(* IEC 61131-3 sources: inproshop/test9_exported/2.Main, 6 files *)

(* ---- Main_Clock.st ---- *)
VAR_GLOBAL
	CPU_Clock:Str_Clock;
END_VAR

(* ---- Main_Communication.st ---- *)
VAR_GLOBAL
	From_OPXX AT %IW2000:Str_OP10_TO_OPXX;
	TO_OPXX AT %QW2000:Str_OPXX_TO_OP10;
	To_Slave:Str_ToSlave;

END_VAR

(* ---- Main_IO.st ---- *)
VAR_GLOBAL

	IX7000_0	AT	%IX7000.0:BOOL;
	IX7000_1	AT	%IX7000.1:BOOL;
	IX7000_2	AT	%IX7000.2:BOOL;
	IX7000_3	AT	%IX7000.3:BOOL;
	IX7000_4	AT	%IX7000.4:BOOL;
	IX7000_5	AT	%IX7000.5:BOOL;
	IX7000_6	AT	%IX7000.6:BOOL;
	IX7000_7	AT	%IX7000.7:BOOL;
	IX7001_0_OP07启动按钮HMI1	AT	%IX7001.0:BOOL;
	IX7001_1_OP07停止按钮HMI1	AT	%IX7001.1:BOOL;
	IX7001_2_OP07复位按钮HMI1	AT	%IX7001.2:BOOL;
	IX7001_3_OP07手自动旋钮HMI1	AT	%IX7001.3:BOOL;
	IX7001_4_OP07急停按钮HMI	AT	%IX7001.4:BOOL;
	IX7001_5_OP07启动按钮左	AT	%IX7001.5:BOOL;
	IX7001_6_OP07停止按钮左	AT	%IX7001.6:BOOL;
	IX7001_7_OP07复位按钮左	AT	%IX7001.7:BOOL;
	IX7002_0_OP07手自动旋钮左	AT	%IX7002.0:BOOL;
	IX7002_1_OP07急停按钮左	AT	%IX7002.1:BOOL;
	IX7002_2_OP07启动按钮右	AT	%IX7002.2:BOOL;
	IX7002_3_OP07停止按钮右	AT	%IX7002.3:BOOL;
	IX7002_4_OP07复位按钮右	AT	%IX7002.4:BOOL;
	IX7002_5_OP07手自动旋钮右	AT	%IX7002.5:BOOL;
	IX7002_6_OP07急停按钮右	AT	%IX7002.6:BOOL;
	IX7002_7_OP07安全门1	AT	%IX7002.7:BOOL;
	IX7003_0_OP07安全门2	AT	%IX7003.0:BOOL;
	IX7003_1_OP07安全门3	AT	%IX7003.1:BOOL;
	IX7003_2_OP07安全门4	AT	%IX7003.2:BOOL;
	IX7003_3_OP07安全门5	AT	%IX7003.3:BOOL;
	IX7003_4_OP07安全门6	AT	%IX7003.4:BOOL;
	IX7003_5_OP07安全门7	AT	%IX7003.5:BOOL;
	IX7003_6_OP07安全门8	AT	%IX7003.6:BOOL;
	IX7003_7	AT	%IX7003.7:BOOL;
	IX7004_0	AT	%IX7004.0:BOOL;
	IX7004_1	AT	%IX7004.1:BOOL;
	IX7004_2	AT	%IX7004.2:BOOL;
	IX7004_3	AT	%IX7004.3:BOOL;
	IX7004_4	AT	%IX7004.4:BOOL;
	IX7004_5	AT	%IX7004.5:BOOL;
	IX7004_6	AT	%IX7004.6:BOOL;
	IX7004_7_水冷机故障	AT	%IX7004.7:BOOL;
	IX7005_0_供钉机1_缺钉报警	AT	%IX7005.0:BOOL;
	IX7005_1_供钉机1_供钉完成	AT	%IX7005.1:BOOL;
	IX7005_2_供钉机1_钉入管检测	AT	%IX7005.2:BOOL;
	IX7005_3_供钉机1_钉到位检测	AT	%IX7005.3:BOOL;
	IX7005_4_电批1_结果OK	AT	%IX7005.4:BOOL;
	IX7005_5_电批1_结果NG	AT	%IX7005.5:BOOL;
	IX7005_6_电批1_ERROR	AT	%IX7005.6:BOOL;
	IX7005_7_电批1_预留	AT	%IX7005.7:BOOL;
	IX7006_0_供钉机2_缺钉报警	AT	%IX7006.0:BOOL;
	IX7006_1_供钉机2_供钉完成	AT	%IX7006.1:BOOL;
	IX7006_2_供钉机2_钉入管检测	AT	%IX7006.2:BOOL;
	IX7006_3_供钉机2_钉到位检测	AT	%IX7006.3:BOOL;
	IX7006_4_电批2_结果OK	AT	%IX7006.4:BOOL;
	IX7006_5_电批2_结果NG	AT	%IX7006.5:BOOL;
	IX7006_6_电批2_ERROR	AT	%IX7006.6:BOOL;
	IX7006_7_电批2_预留	AT	%IX7006.7:BOOL;
	IX7007_0_供钉机3_缺钉报警	AT	%IX7007.0:BOOL;
	IX7007_1_供钉机3_供钉完成	AT	%IX7007.1:BOOL;
	IX7007_2_供钉机3_钉入管检测	AT	%IX7007.2:BOOL;
	IX7007_3_供钉机3_钉到位检测	AT	%IX7007.3:BOOL;
	IX7007_4_电批3_结果OK	AT	%IX7007.4:BOOL;
	IX7007_5_电批3_结果NG	AT	%IX7007.5:BOOL;
	IX7007_6_电批3_ERROR	AT	%IX7007.6:BOOL;
	IX7007_7_电批3_预留	AT	%IX7007.7:BOOL;
	IX7008_0_供钉机4_供钉完成	AT	%IX7008.0:BOOL;
	IX7008_1_供钉机4_预留	AT	%IX7008.1:BOOL;
	IX7008_2_供钉机4_预留	AT	%IX7008.2:BOOL;
	IX7008_3_供钉机4_预留	AT	%IX7008.3:BOOL;
	IX7008_4_电批4_结果OK	AT	%IX7008.4:BOOL;
	IX7008_5_电批4_结果NG	AT	%IX7008.5:BOOL;
	IX7008_6_电批4_ERROR	AT	%IX7008.6:BOOL;
	IX7008_7_电批4_预留	AT	%IX7008.7:BOOL;
	IX7009_0	AT	%IX7009.0:BOOL;
	IX7009_1	AT	%IX7009.1:BOOL;
	IX7009_2	AT	%IX7009.2:BOOL;
	IX7009_3	AT	%IX7009.3:BOOL;
	IX7009_4	AT	%IX7009.4:BOOL;
	IX7009_5	AT	%IX7009.5:BOOL;
	IX7009_6	AT	%IX7009.6:BOOL;
	IX7009_7	AT	%IX7009.7:BOOL;
	IX7100_0_启动按钮1	AT	%IX7100.0:BOOL;
	IX7100_1_启动按钮2	AT	%IX7100.1:BOOL;
	IX7100_2_安全光栅	AT	%IX7100.2:BOOL;
	IX7100_3	AT	%IX7100.3:BOOL;
	IX7100_4_上料1侧边定位气缸CY01_伸出	AT	%IX7100.4:BOOL;
	IX7100_5_上料1侧边定位气缸CY01_缩回	AT	%IX7100.5:BOOL;
	IX7100_6_上料避位升降气缸CY02_上升	AT	%IX7100.6:BOOL;
	IX7100_7_上料避位升降气缸CY02_下降	AT	%IX7100.7:BOOL;
	IX7101_0_物料有无检测Sensor1	AT	%IX7101.0:BOOL;
	IX7101_1_物料有无检测Sensor2	AT	%IX7101.1:BOOL;
	IX7101_2	AT	%IX7101.2:BOOL;
	IX7101_3	AT	%IX7101.3:BOOL;
	IX7101_4	AT	%IX7101.4:BOOL;
	IX7101_5	AT	%IX7101.5:BOOL;
	IX7101_6	AT	%IX7101.6:BOOL;
	IX7101_7	AT	%IX7101.7:BOOL;
	IX7102_0_搬运1_1旋转气缸CY03_放料位	AT	%IX7102.0:BOOL;
	IX7102_1_搬运1_1旋转气缸CY03_取料位	AT	%IX7102.1:BOOL;
	IX7102_2_搬运1_1夹爪气缸CY04_夹紧位	AT	%IX7102.2:BOOL;
	IX7102_3_搬运1_1夹爪气缸CY04_打开位	AT	%IX7102.3:BOOL;
	IX7102_4_搬运1_1避让气缸CY05A_伸出位	AT	%IX7102.4:BOOL;
	IX7102_5_搬运1_1避让气缸CY05A_缩回位	AT	%IX7102.5:BOOL;
	IX7102_6_搬运1_1避让气缸CY05B_伸出位	AT	%IX7102.6:BOOL;
	IX7102_7_搬运1_1避让气缸CY05B_缩回位	AT	%IX7102.7:BOOL;
	IX7103_0_搬运1_2旋转气缸CY06_放料位	AT	%IX7103.0:BOOL;
	IX7103_1_搬运1_2旋转气缸CY06_取料位	AT	%IX7103.1:BOOL;
	IX7103_2_搬运1_2夹爪气缸CY07_夹紧位	AT	%IX7103.2:BOOL;
	IX7103_3_搬运1_2夹爪气缸CY07_打开位	AT	%IX7103.3:BOOL;
	IX7103_4_搬运1_2避让气缸CY08_伸出位	AT	%IX7103.4:BOOL;
	IX7103_5_搬运1_2避让气缸CY08_缩回位	AT	%IX7103.5:BOOL;
	IX7103_6	AT	%IX7103.6:BOOL;
	IX7103_7	AT	%IX7103.7:BOOL;
	IX7104_0_搬运2_1旋转气缸CY09_放料位	AT	%IX7104.0:BOOL;
	IX7104_1_搬运2_1旋转气缸CY09_取料位	AT	%IX7104.1:BOOL;
	IX7104_2_搬运2_1夹爪气缸CY10_夹紧位	AT	%IX7104.2:BOOL;
	IX7104_3_搬运2_1夹爪气缸CY10_打开位	AT	%IX7104.3:BOOL;
	IX7104_4_搬运2_1避让气缸CY11_伸出位	AT	%IX7104.4:BOOL;
	IX7104_5_搬运2_1避让气缸CY11_缩回位	AT	%IX7104.5:BOOL;
	IX7104_6	AT	%IX7104.6:BOOL;
	IX7104_7	AT	%IX7104.7:BOOL;
	IX7105_0_搬运2_2旋转气缸CY12_放料位	AT	%IX7105.0:BOOL;
	IX7105_1_搬运2_2旋转气缸CY12_取料位	AT	%IX7105.1:BOOL;
	IX7105_2_搬运2_2夹爪气缸CY13_夹紧位	AT	%IX7105.2:BOOL;
	IX7105_3_搬运2_2夹爪气缸CY13_打开位	AT	%IX7105.3:BOOL;
	IX7105_4_搬运2_2避让气缸CY14_伸出位	AT	%IX7105.4:BOOL;
	IX7105_5_搬运2_2避让气缸CY14_缩回位	AT	%IX7105.5:BOOL;
	IX7105_6	AT	%IX7105.6:BOOL;
	IX7105_7	AT	%IX7105.7:BOOL;
	IX7106_0_平台1避位升降气缸CY15_上升位	AT	%IX7106.0:BOOL;
	IX7106_1_平台1避位升降气缸CY15_下降位	AT	%IX7106.1:BOOL;
	IX7106_2_平台1侧推定位X气缸CY16_缩回位	AT	%IX7106.2:BOOL;
	IX7106_3_平台1侧推定位X气缸CY16_伸出位	AT	%IX7106.3:BOOL;
	IX7106_4_平台1侧推定位Y气缸CY17_伸出位	AT	%IX7106.4:BOOL;
	IX7106_5_平台1侧推定位Y气缸CY17_缩回位	AT	%IX7106.5:BOOL;
	IX7106_6_平台1物料压紧气缸CY18_下降位	AT	%IX7106.6:BOOL;
	IX7106_7_平台1物料压紧气缸CY18_上升位	AT	%IX7106.7:BOOL;
	IX7107_0_平台1物料有无检测Sensor3	AT	%IX7107.0:BOOL;
	IX7107_1_平台2物料有无检测Sensor4	AT	%IX7107.1:BOOL;
	IX7107_2_平台2避位升降气缸CY19_上升位	AT	%IX7107.2:BOOL;
	IX7107_3_平台2避位升降气缸CY19_下降位	AT	%IX7107.3:BOOL;
	IX7107_4_平台2侧推定位Y气缸CY20_伸出位	AT	%IX7107.4:BOOL;
	IX7107_5_平台2侧推定位Y气缸CY20_缩回位	AT	%IX7107.5:BOOL;
	IX7107_6_平台2物料压紧气缸CY21_下降位	AT	%IX7107.6:BOOL;
	IX7107_7_平台2物料压紧气缸CY21_上升位	AT	%IX7107.7:BOOL;
	IX7108_0_平台3避位升降气缸CY22_上升位	AT	%IX7108.0:BOOL;
	IX7108_1_平台3避位升降气缸CY22_下降位	AT	%IX7108.1:BOOL;
	IX7108_2_平台4侧推定位X气缸CY23_缩回位	AT	%IX7108.2:BOOL;
	IX7108_3_平台4侧推定位X气缸CY23_伸出位	AT	%IX7108.3:BOOL;
	IX7108_4_平台3侧推定位Y气缸CY24_伸出位	AT	%IX7108.4:BOOL;
	IX7108_5_平台3侧推定位Y气缸CY24_缩回位	AT	%IX7108.5:BOOL;
	IX7108_6_平台3物料压紧气缸CY25_下降位	AT	%IX7108.6:BOOL;
	IX7108_7_平台3物料压紧气缸CY25_上升位	AT	%IX7108.7:BOOL;
	IX7109_0_平台3物料有无检测Sensor5	AT	%IX7109.0:BOOL;
	IX7109_1_平台4物料有无检测Sensor6	AT	%IX7109.1:BOOL;
	IX7109_2_平台4避位升降气缸CY26_上升位	AT	%IX7109.2:BOOL;
	IX7109_3_平台4避位升降气缸CY26_下降位	AT	%IX7109.3:BOOL;
	IX7109_4_平台4侧推定位Y气缸CY27_缩回位	AT	%IX7109.4:BOOL;
	IX7109_5_平台4侧推定位Y气缸CY27_伸出位	AT	%IX7109.5:BOOL;
	IX7109_6_平台4物料旋转气缸CY28_下料位	AT	%IX7109.6:BOOL;
	IX7109_7_平台4物料旋转气缸CY28_接料位	AT	%IX7109.7:BOOL;
	IX7110_0_电批1上下气缸CY30_下降位	AT	%IX7110.0:BOOL;
	IX7110_1_电批1上下气缸CY30_上升位	AT	%IX7110.1:BOOL;
	IX7110_2_电批2上下气缸CY31_下降位	AT	%IX7110.2:BOOL;
	IX7110_3_电批2上下气缸CY31_上升位	AT	%IX7110.3:BOOL;
	IX7110_4	AT	%IX7110.4:BOOL;
	IX7110_5	AT	%IX7110.5:BOOL;
	IX7110_6_电批3整体上下气缸CY32_下降位	AT	%IX7110.6:BOOL;
	IX7110_7_电批3整体上下气缸CY32_上升位	AT	%IX7110.7:BOOL;
	IX7111_0_电批3鸟嘴上下气缸CY33_下降位	AT	%IX7111.0:BOOL;
	IX7111_1_电批3鸟嘴上下气缸CY33_上升位	AT	%IX7111.1:BOOL;
	IX7111_2_电批3真空Vac01_真空表头	AT	%IX7111.2:BOOL;
	IX7111_3	AT	%IX7111.3:BOOL;
	IX7111_4_电批4上下气缸CY34_下降位	AT	%IX7111.4:BOOL;
	IX7111_5_电批4上下气缸CY34_上升位	AT	%IX7111.5:BOOL;
	IX7111_6_电批4真空Vac02_真空表头	AT	%IX7111.6:BOOL;
	IX7111_7	AT	%IX7111.7:BOOL;
	QX7000_0	AT	%QX7000.0:BOOL;
	QX7000_1	AT	%QX7000.1:BOOL;
	QX7000_2	AT	%QX7000.2:BOOL;
	QX7000_3	AT	%QX7000.3:BOOL;
	QX7000_4	AT	%QX7000.4:BOOL;
	QX7000_5	AT	%QX7000.5:BOOL;
	QX7000_6	AT	%QX7000.6:BOOL;
	QX7000_7	AT	%QX7000.7:BOOL;
	QX7001_0_OP07启动按钮指示灯HMI	AT	%QX7001.0:BOOL;
	QX7001_1_OP07停止按钮指示灯HMI	AT	%QX7001.1:BOOL;
	QX7001_2_OP07复位按钮指示灯HMI	AT	%QX7001.2:BOOL;
	QX7001_3_OP07启动按钮指示灯左	AT	%QX7001.3:BOOL;
	QX7001_4_OP07停止按钮指示灯左	AT	%QX7001.4:BOOL;
	QX7001_5_OP07复位按钮指示灯左	AT	%QX7001.5:BOOL;
	QX7001_6_OP07启动按钮指示灯右	AT	%QX7001.6:BOOL;
	QX7001_7_OP07停止按钮指示灯右	AT	%QX7001.7:BOOL;
	QX7002_0_OP07复位按钮指示灯右	AT	%QX7002.0:BOOL;
	QX7002_1_OP07三色灯红	AT	%QX7002.1:BOOL;
	QX7002_2_OP07三色灯黄	AT	%QX7002.2:BOOL;
	QX7002_3_OP07三色灯绿	AT	%QX7002.3:BOOL;
	QX7002_4_OP07蜂鸣器	AT	%QX7002.4:BOOL;
	QX7002_5_OP07照明灯	AT	%QX7002.5:BOOL;
	QX7002_6	AT	%QX7002.6:BOOL;
	QX7002_7	AT	%QX7002.7:BOOL;
	QX7003_0	AT	%QX7003.0:BOOL;
	QX7003_1	AT	%QX7003.1:BOOL;
	QX7003_2	AT	%QX7003.2:BOOL;
	QX7003_3	AT	%QX7003.3:BOOL;
	QX7003_4	AT	%QX7003.4:BOOL;
	QX7003_5	AT	%QX7003.5:BOOL;
	QX7003_6	AT	%QX7003.6:BOOL;
	QX7003_7	AT	%QX7003.7:BOOL;
	QX7004_0	AT	%QX7004.0:BOOL;
	QX7004_1	AT	%QX7004.1:BOOL;
	QX7004_2	AT	%QX7004.2:BOOL;
	QX7004_3	AT	%QX7004.3:BOOL;
	QX7004_4	AT	%QX7004.4:BOOL;
	QX7004_5	AT	%QX7004.5:BOOL;
	QX7004_6	AT	%QX7004.6:BOOL;
	QX7004_7	AT	%QX7004.7:BOOL;
	QX7005_0_供钉机1_启动供钉	AT	%QX7005.0:BOOL;
	QX7005_1_供钉机1_预留	AT	%QX7005.1:BOOL;
	QX7005_2_供钉机1_预留	AT	%QX7005.2:BOOL;
	QX7005_3_供钉机1_预留	AT	%QX7005.3:BOOL;
	QX7005_4_电批1_使能	AT	%QX7005.4:BOOL;
	QX7005_5_电批1_启动	AT	%QX7005.5:BOOL;
	QX7005_6_电批1_预留	AT	%QX7005.6:BOOL;
	QX7005_7_电批1_预留	AT	%QX7005.7:BOOL;
	QX7006_0_供钉机2_启动供钉	AT	%QX7006.0:BOOL;
	QX7006_1_供钉机2_预留	AT	%QX7006.1:BOOL;
	QX7006_2_供钉机2_预留	AT	%QX7006.2:BOOL;
	QX7006_3_供钉机2_预留	AT	%QX7006.3:BOOL;
	QX7006_4_电批2_使能	AT	%QX7006.4:BOOL;
	QX7006_5_电批2_启动	AT	%QX7006.5:BOOL;
	QX7006_6_电批2_预留	AT	%QX7006.6:BOOL;
	QX7006_7_电批2_预留	AT	%QX7006.7:BOOL;
	QX7007_0_供钉机3_启动供钉	AT	%QX7007.0:BOOL;
	QX7007_1_供钉机3_预留	AT	%QX7007.1:BOOL;
	QX7007_2_供钉机3_预留	AT	%QX7007.2:BOOL;
	QX7007_3_供钉机3_预留	AT	%QX7007.3:BOOL;
	QX7007_4_电批3_使能	AT	%QX7007.4:BOOL;
	QX7007_5_电批3_启动	AT	%QX7007.5:BOOL;
	QX7007_6_电批3_预留	AT	%QX7007.6:BOOL;
	QX7007_7_电批3_预留	AT	%QX7007.7:BOOL;
	QX7008_0_供钉机4_启动供钉	AT	%QX7008.0:BOOL;
	QX7008_1_供钉机4_预留	AT	%QX7008.1:BOOL;
	QX7008_2_供钉机4_预留	AT	%QX7008.2:BOOL;
	QX7008_3_供钉机4_预留	AT	%QX7008.3:BOOL;
	QX7008_4_电批4_使能	AT	%QX7008.4:BOOL;
	QX7008_5_电批4_启动	AT	%QX7008.5:BOOL;
	QX7008_6_电批4_预留	AT	%QX7008.6:BOOL;
	QX7008_7_电批4_预留	AT	%QX7008.7:BOOL;
	QX7009_0	AT	%QX7009.0:BOOL;
	QX7009_1	AT	%QX7009.1:BOOL;
	QX7009_2	AT	%QX7009.2:BOOL;
	QX7009_3	AT	%QX7009.3:BOOL;
	QX7009_4	AT	%QX7009.4:BOOL;
	QX7009_5	AT	%QX7009.5:BOOL;
	QX7009_6	AT	%QX7009.6:BOOL;
	QX7009_7	AT	%QX7009.7:BOOL;
	QX7100_0_启动按钮1指示灯	AT	%QX7100.0:BOOL;
	QX7100_1_启动按钮2指示灯	AT	%QX7100.1:BOOL;
	QX7100_2	AT	%QX7100.2:BOOL;
	QX7100_3	AT	%QX7100.3:BOOL;
	QX7100_4_上料1侧边定位气缸CY01_伸出	AT	%QX7100.4:BOOL;
	QX7100_5_上料1侧边定位气缸CY01_缩回	AT	%QX7100.5:BOOL;
	QX7100_6_上料避位升降气缸CY02_上升	AT	%QX7100.6:BOOL;
	QX7100_7_上料避位升降气缸CY02_下降	AT	%QX7100.7:BOOL;
	QX7101_0	AT	%QX7101.0:BOOL;
	QX7101_1	AT	%QX7101.1:BOOL;
	QX7101_2	AT	%QX7101.2:BOOL;
	QX7101_3	AT	%QX7101.3:BOOL;
	QX7101_4	AT	%QX7101.4:BOOL;
	QX7101_5	AT	%QX7101.5:BOOL;
	QX7101_6	AT	%QX7101.6:BOOL;
	QX7101_7	AT	%QX7101.7:BOOL;
	QX7102_0_搬运1_1旋转气缸CY03_放料	AT	%QX7102.0:BOOL;
	QX7102_1_搬运1_1旋转气缸CY03_取料	AT	%QX7102.1:BOOL;
	QX7102_2_搬运1_1夹爪气缸CY04_夹紧	AT	%QX7102.2:BOOL;
	QX7102_3_搬运1_1夹爪气缸CY04_打开	AT	%QX7102.3:BOOL;
	QX7102_4_搬运1_1避让气缸CY05_伸出	AT	%QX7102.4:BOOL;
	QX7102_5_搬运1_1避让气缸CY05_缩回	AT	%QX7102.5:BOOL;
	QX7102_6	AT	%QX7102.6:BOOL;
	QX7102_7	AT	%QX7102.7:BOOL;
	QX7103_0_搬运1_2旋转气缸CY06_放料	AT	%QX7103.0:BOOL;
	QX7103_1_搬运1_2旋转气缸CY06_取料	AT	%QX7103.1:BOOL;
	QX7103_2_搬运1_2夹爪气缸CY07_夹紧	AT	%QX7103.2:BOOL;
	QX7103_3_搬运1_2夹爪气缸CY07_打开	AT	%QX7103.3:BOOL;
	QX7103_4_搬运1_2避让气缸CY08_伸出	AT	%QX7103.4:BOOL;
	QX7103_5_搬运1_2避让气缸CY08_缩回	AT	%QX7103.5:BOOL;
	QX7103_6	AT	%QX7103.6:BOOL;
	QX7103_7	AT	%QX7103.7:BOOL;
	QX7104_0_搬运2_1旋转气缸CY09_放料	AT	%QX7104.0:BOOL;
	QX7104_1_搬运2_1旋转气缸CY09_取料	AT	%QX7104.1:BOOL;
	QX7104_2_搬运2_1夹爪气缸CY10_夹紧	AT	%QX7104.2:BOOL;
	QX7104_3_搬运2_1夹爪气缸CY10_打开	AT	%QX7104.3:BOOL;
	QX7104_4_搬运2_1避让气缸CY11_伸出	AT	%QX7104.4:BOOL;
	QX7104_5_搬运2_1避让气缸CY11_缩回	AT	%QX7104.5:BOOL;
	QX7104_6	AT	%QX7104.6:BOOL;
	QX7104_7	AT	%QX7104.7:BOOL;
	QX7105_0_搬运2_2旋转气缸CY12_放料	AT	%QX7105.0:BOOL;
	QX7105_1_搬运2_2旋转气缸CY12_取料	AT	%QX7105.1:BOOL;
	QX7105_2_搬运2_2夹爪气缸CY13_夹紧	AT	%QX7105.2:BOOL;
	QX7105_3_搬运2_2夹爪气缸CY13_打开	AT	%QX7105.3:BOOL;
	QX7105_4_搬运2_2避让气缸CY14_伸出	AT	%QX7105.4:BOOL;
	QX7105_5_搬运2_2避让气缸CY14_缩回	AT	%QX7105.5:BOOL;
	QX7105_6	AT	%QX7105.6:BOOL;
	QX7105_7	AT	%QX7105.7:BOOL;
	QX7106_0_平台1避升降气缸CY15_上升	AT	%QX7106.0:BOOL;
	QX7106_1_平台1避升降气缸CY15_下降	AT	%QX7106.1:BOOL;
	QX7106_2_平台1侧推定X气缸CY16_缩回	AT	%QX7106.2:BOOL;
	QX7106_3_平台1侧推定X气缸CY16_伸出	AT	%QX7106.3:BOOL;
	QX7106_4_平台1侧推定Y气缸CY17_伸出	AT	%QX7106.4:BOOL;
	QX7106_5_平台1侧推定Y气缸CY17_缩回	AT	%QX7106.5:BOOL;
	QX7106_6_平台1物料压紧气缸CY18_下降	AT	%QX7106.6:BOOL;
	QX7106_7_平台1物料压紧气缸CY18_上升	AT	%QX7106.7:BOOL;
	QX7107_0	AT	%QX7107.0:BOOL;
	QX7107_1	AT	%QX7107.1:BOOL;
	QX7107_2_平台2避升降气缸CY19_上升	AT	%QX7107.2:BOOL;
	QX7107_3_平台2避升降气缸CY19_下降	AT	%QX7107.3:BOOL;
	QX7107_4_平台2侧推定Y气缸CY20_伸出	AT	%QX7107.4:BOOL;
	QX7107_5_平台2侧推定Y气缸CY20_缩回	AT	%QX7107.5:BOOL;
	QX7107_6_平台2物料压紧气缸CY21_下降	AT	%QX7107.6:BOOL;
	QX7107_7_平台2物料压紧气缸CY21_上升	AT	%QX7107.7:BOOL;
	QX7108_0_平台3避升降气缸CY22_上升	AT	%QX7108.0:BOOL;
	QX7108_1_平台3避升降气缸CY22_下降	AT	%QX7108.1:BOOL;
	QX7108_2_平台4侧推定X气缸CY23_缩回	AT	%QX7108.2:BOOL;
	QX7108_3_平台4侧推定X气缸CY23_伸出	AT	%QX7108.3:BOOL;
	QX7108_4_平台3侧推定Y气缸CY24_伸出	AT	%QX7108.4:BOOL;
	QX7108_5_平台3侧推定Y气缸CY24_缩回	AT	%QX7108.5:BOOL;
	QX7108_6_平台3物料压紧气缸CY25_下降	AT	%QX7108.6:BOOL;
	QX7108_7_平台3物料压紧气缸CY25_上升	AT	%QX7108.7:BOOL;
	QX7109_0	AT	%QX7109.0:BOOL;
	QX7109_1	AT	%QX7109.1:BOOL;
	QX7109_2_平台4避升降气缸CY26_上升	AT	%QX7109.2:BOOL;
	QX7109_3_平台4避升降气缸CY26_下降	AT	%QX7109.3:BOOL;
	QX7109_4_平台4侧推定Y气缸CY27_缩回	AT	%QX7109.4:BOOL;
	QX7109_5_平台4侧推定Y气缸CY27_伸出	AT	%QX7109.5:BOOL;
	QX7109_6_平台4物料压紧气缸CY28_下料	AT	%QX7109.6:BOOL;
	QX7109_7_平台4物料压紧气缸CY28_接料	AT	%QX7109.7:BOOL;
	QX7110_0_电批1上下气缸CY30_下降	AT	%QX7110.0:BOOL;
	QX7110_1_电批1上下气缸CY30_上升	AT	%QX7110.1:BOOL;
	QX7110_2_电批2上下气缸CY31_下降	AT	%QX7110.2:BOOL;
	QX7110_3_电批2上下气缸CY31_上升	AT	%QX7110.3:BOOL;
	QX7110_4	AT	%QX7110.4:BOOL;
	QX7110_5	AT	%QX7110.5:BOOL;
	QX7110_6_电批3整体上下气缸CY32_下降	AT	%QX7110.6:BOOL;
	QX7110_7_电批3整体上下气缸CY32_上升	AT	%QX7110.7:BOOL;
	QX7111_0_电批3鸟嘴上下气缸CY33_下降	AT	%QX7111.0:BOOL;
	QX7111_1_电批3鸟嘴上下气缸CY33_上升	AT	%QX7111.1:BOOL;
	QX7111_2_电批3真空Vac01_吸真空	AT	%QX7111.2:BOOL;
	QX7111_3_电批3真空Vac01_破真空	AT	%QX7111.3:BOOL;
	QX7111_4_电批4上下气缸CY34_下降	AT	%QX7111.4:BOOL;
	QX7111_5_电批4上下气缸CY34_上升	AT	%QX7111.5:BOOL;
	QX7111_6_电批4真空Vac02_吸真空	AT	%QX7111.6:BOOL;
	QX7111_7_电批4真空Vac02_破真空	AT	%QX7111.7:BOOL;
END_VAR

VAR_GLOBAL

END_VAR

(* ---- Clock.st ---- *)
PROGRAM Clock
VAR
	data_clock_10ms:FB_Clock;
	data_clock_50ms:FB_Clock;
	data_clock_100ms:FB_Clock;
	data_clock_500ms:FB_Clock;
	data_clock_1s:FB_Clock;
END_VAR

//100MS脉冲
data_clock_10ms(iEnable:=TRUE,iClock:=1,o_Clock=>CPU_Clock.Clock_10ms);

//500MS脉冲
data_clock_50ms(iEnable:=TRUE,iClock:=5,o_Clock=>CPU_Clock.Clock_50ms);

//100MS脉冲
data_clock_100ms(iEnable:=TRUE,iClock:=10,o_Clock=>CPU_Clock.Clock_100ms);

//500MS脉冲
data_clock_500ms(iEnable:=TRUE,iClock:=50,o_Clock=>CPU_Clock.Clock_500ms);

//1S脉冲
data_clock_1s(iEnable:=TRUE,iClock:=100,o_Clock=>CPU_Clock.Clock_1s);

(* ---- PLC_PRG.st ---- *)
PROGRAM PLC_PRG
VAR
	Temp_pulse_on_R:R_TRIG;
	Temp_clock_10ms_R:R_TRIG;
	Temp_clock_50ms_R:R_TRIG;
	Temp_clock_100ms_R:R_TRIG;
	Temp_clock_500ms_R:R_TRIG;
	Temp_clock_1s_R:R_TRIG;

END_VAR
//RUN之后一个扫描周期ON
Temp_pulse_on_R(CLK:=TRUE,Q=>CPU_Clock.FirstRun);

//10ms脉冲上升沿
Temp_clock_10ms_R(CLK:=CPU_Clock.Clock_10ms,Q=>CPU_Clock.Clock_10ms_R);

//50ms脉冲上升沿
Temp_clock_50ms_R(CLK:=CPU_Clock.Clock_50ms,Q=>CPU_Clock.Clock_50ms_R);

//100ms脉冲上升沿
Temp_clock_100ms_R(CLK:=CPU_Clock.Clock_100ms,Q=>CPU_Clock.Clock_100ms_R);

//500ms脉冲上升沿
Temp_clock_500ms_R(CLK:=CPU_Clock.Clock_500ms,Q=>CPU_Clock.Clock_500ms_R);

//1s脉冲上升沿
Temp_clock_1s_R(CLK:=CPU_Clock.Clock_1s,Q=>CPU_Clock.Clock_1s_R);

//累计运行时间ms获取
GetSystemTime(udiTimeMs=>CPU_Clock.TimeMs );
//获取系统时间
GetSystemDate_sDt(stSystemDate=>CPU_Clock.DataToday);
//获取前31天时间
FC_SysTime(iNow:= CPU_Clock.DataToday, ioBefor:=CPU_Clock.DateOld );

//开班时间设定
CPU_Clock.DayStartTime:='8:30';
CPU_Clock.NightStartTime:='20:30';
//

OP10_Control();
OP11_Control();
OP20_Control();
OP30_Control();
OP70_Control();
OP80_Control();

(* ---- Test.st ---- *)
PROGRAM Test

VAR

	i:INT;
	PickPoint:INT;
END_VAR
